(* IEC 61131-3 sources: AXOpen/src/components.dukane.welders/ctrl/src/Axo_IQ_SeriesWelder/TypesStructuresAndEnums, 6 files *)

(* ---- Axo_IQ_SeriesWelder_Config.st ---- *)
NAMESPACE AXOpen.Components.Dukane.Welders
    {S7.extern=ReadWrite}
    {#ix-attr:[Container(Layout.Stack)]}
    CLASS PUBLIC Axo_IQ_SeriesWelder_Config
        VAR PUBLIC
            {#ix-set:AttributeName = "<#Info time#>"}
            InfoTime : LTIME := LT#5S;
            {#ix-set:AttributeName = "<#Error time#>"}
            ErrorTime : LTIME := LT#10S;
            {#ix-set:AttributeName = "<#Task timeout#>"}
            TaskTimeout : LTIME := LT#50S;
            {#ix-set:AttributeName = "<#Hardware IDs#>"}
            HWIDs : Axo_IQ_SeriesWelder_HWIDs;
        END_VAR
    END_CLASS
END_NAMESPACE

(* ---- Axo_IQ_SeriesWelder_Control.st ---- *)
NAMESPACE AXOpen.Components.Dukane.Welders
    {S7.extern=ReadWrite}
    {#ix-attr:[Container(Layout.Stack)]}
    CLASS PUBLIC Axo_IQ_SeriesWelder_Control
        VAR PUBLIC

        END_VAR
    END_CLASS
END_NAMESPACE

(* ---- Axo_IQ_SeriesWelder_HWIDs.st ---- *)
NAMESPACE AXOpen.Components.Dukane.Welders
   {S7.extern=ReadWrite}
	CLASS Axo_IQ_SeriesWelder_HWIDs
      VAR PUBLIC
         {#ix-set:AttributeName = "<#Hardware ID  of the device#>"}
         HW_Device              :  UINT;
         {#ix-set:AttributeName = "<#Hardware ID of the 'iQ_to_PLC_Inputs' submodule#>"}
         HwID_iQ_to_PLC_Inputs  :   UINT;
         {#ix-set:AttributeName = "<#Hardware ID of the 'out_1' submodule#>"}
         HwID_PLC_to_iQ_Outputs           :   UINT;
      END_VAR
   END_CLASS
END_NAMESPACE

(* ---- Axo_IQ_SeriesWelder_In.st ---- *)
NAMESPACE AXOpen.Components.Dukane.Welders
    {S7.extern=ReadWrite}
    {#ix-attr:[Container(Layout.Wrap)]}
    CLASS PUBLIC Axo_IQ_SeriesWelder_In
        VAR PUBLIC
            {#ix-set:AttributeName = "<#Status#>"}
            {#ix-attr:[ReadOnly()]}
            Status           :   Axo_IQ_SeriesWelder_Status;
        END_VAR
    END_CLASS
END_NAMESPACE

(* ---- Axo_IQ_SeriesWelder_Out.st ---- *)
NAMESPACE AXOpen.Components.Dukane.Welders
    {S7.extern=ReadWrite}
    {#ix-attr:[Container(Layout.Wrap)]}
    CLASS PUBLIC Axo_IQ_SeriesWelder_Out
        VAR PUBLIC
            {#ix-set:AttributeName = "<#Control#>"}
            {#ix-attr:[ReadOnly()]}
            Control           :   Axo_IQ_SeriesWelder_Control;
        END_VAR
    END_CLASS
END_NAMESPACE

(* ---- Axo_IQ_SeriesWelder_Status.st ---- *)
NAMESPACE AXOpen.Components.Dukane.Welders
    {S7.extern=ReadWrite}
    {#ix-attr:[Container(Layout.Stack)]}
    CLASS PUBLIC Axo_IQ_SeriesWelder_Status
        VAR PUBLIC

        END_VAR
    END_CLASS
END_NAMESPACE
